// TwinCAT 3 PLC project RedLine3
// ProgramVersion: 3.1.4023.0
// libraries:
//   Tc2_Standard, * (Beckhoff Automation GmbH)
//   Tc2_System, * (Beckhoff Automation GmbH)
//   Tc3_Module, * (Beckhoff Automation GmbH)
// project tree:
//   GVLs/ GVL.TcGVL
//   / PlcTask.TcTTO
//   POUs/ MAIN.TcPOU

CONFIGURATION RedLine3
    RESOURCE PLC ON TwinCAT3
        TASK PlcTask(INTERVAL := T#10ms, PRIORITY := 20);
        PROGRAM MAIN WITH PlcTask : MAIN;
    END_RESOURCE
END_CONFIGURATION

// ---- GVLs/GVL.TcGVL
{attribute 'qualified_only'}
VAR_GLOBAL

//Block States IO
mInSwitch : ARRAY[0..44] OF DINT;
mOutSwitch : ARRAY[0..44] OF DINT;
mInOccupancies : ARRAY[0..44] OF DINT;
mOutOccupancies : ARRAY[0..44] OF DINT;
mInSpeeds : ARRAY[0..44] OF DINT;
mOutSpeeds : ARRAY[0..44] OF DINT;
mInAuthorities : ARRAY[0..44] OF DINT;
mOutAuthorities : ARRAY[0..44] OF DINT;
mInCrossings : ARRAY[0..44] OF DINT;
mOutCrossings : ARRAY[0..44] OF DINT;
mInLeftLights : ARRAY[0..44] OF DINT;
mOutLeftLights : ARRAY[0..44] OF DINT;
mInRightLights : ARRAY[0..44] OF DINT;
mOutRightLights : ARRAY[0..44] OF DINT;
mInMaintenance : ARRAY[0..44] OF DINT;
mOutMaintenance : ARRAY[0..44] OF DINT;
mSpeedLimits : ARRAY[0..44] OF DINT := [40,40,40,40,40,40,40,40,40,40,40,40,40,40,40,40,55,70,70,70,55,55,55,70,70,70,70,70,70,70,70,70,70,70,70,70,70,70,55,55,55,55,55,70];
mInRoute : ARRAY[0..76] OF DINT;
mOutRoute : ARRAY[0..76] OF DINT;


END_VAR

// ---- POUs/MAIN.TcPOU
PROGRAM MAIN
VAR

inc1 : DINT := 0;

	
END_VAR

//0 to 37 map to blocks 1-38
//39 to 44 map to 72-76,yard
//Lights Logic
FOR inc1 := 0 TO 44 DO
	//Sets Red Lights
	IF GVL.mInOccupancies[inc1] = 0
	THEN
		GVL.mOutLeftLights[inc1] := 0;
		GVL.mOutRightLights[inc1] := 0;
	//Sets green lights
	ELSE
		GVL.mOutLeftLights[inc1] := 2;
		GVL.mOutRightLights[inc1] := 2;
	END_IF
END_FOR

FOR inc1 := 1 TO 43 DO
	//Sets Yellow Lights
	IF GVL.mInOccupancies[inc1-1] = 0 AND GVL.mInOccupancies[inc1] <> 0
	THEN
		GVL.mOutRightLights[inc1] := 1;
	END_IF
	IF GVL.mInOccupancies[inc1+1] = 0 AND GVL.mInOccupancies[inc1] <> 0
	THEN
	GVL.mOutLeftLights[inc1] := 1;
	END_IF
END_FOR

//0 to 37 map to blocks 1-38
//39 to 44 map to blocks 72-76,yard
//Passes occupancy, authority, maintenance, and speeds from input to output.
FOR inc1 := 0 TO 44 DO

	GVL.mOutOccupancies[inc1] := GVL.mInOccupancies[inc1];
	GVL.mOutAuthorities[inc1] := GVL.mInAuthorities[inc1];
	GVL.mOutMaintenance[inc1] := GVL.mInMaintenance[inc1];
	IF GVL.mInSpeeds[inc1] < GVL.mSpeedLimits[inc1]
	THEN
		GVL.mOutSpeeds[inc1] := GVL.mInSpeeds[inc1];
	ELSE
		GVL.mOutSpeeds[inc1] := GVL.mSpeedLimits[inc1];
	END_IF
	
END_FOR

FOR inc1 := 0 TO 44 DO

	GVL.mOutRoute[inc1] := GVL.mInRoute[inc1];
	
END_FOR

inc1 := 0;

//This starts the main track logic section

//0 to 37 map to blocks 1-38
//39 to 44 map to 72-76,yard
//Switch Logic
IF GVL.mInMaintenance[8] = 1 
THEN
	IF GVL.mInSwitch[8] = 1
	THEN
		IF GVL.mOutSwitch[8] = 76
		THEN
			GVL.mOutSwitch[8] := 9;
		ELSE
			GVL.mOutSwitch[8] := 76;
		END_IF
		GVL.mInSwitch[8] := 0;
	END_IF
ELSE
    IF GVL.mInOccupancies[44] = 0 
	THEN
    	GVL.mOutSwitch[8] := 76;
    ELSE
		GVL.mOutSwitch[8] := 9;
	END_IF
END_IF

//0 to 37 map to blocks 1-38
//39 to 44 map to 72-76,yard
IF GVL.mInMaintenance[15] = 1 
THEN
    IF GVL.mInSwitch[15] = 1
	THEN
		IF GVL.mOutSwitch[15] = 0
		THEN
			GVL.mOutSwitch[15] := 14;
		ELSE
			GVL.mOutSwitch[15] := 0;
		END_IF
		GVL.mInSwitch[15] := 0;
	END_IF
ELSE
    IF GVL.mInOccupancies[14] = 0 
	THEN
    FOR inc1 := 16 TO 26 DO 
        IF GVL.mInOccupancies[inc1] = 0 
		THEN
            GVL.mOutSwitch[15] := 14;
            Exit;
        ELSE 
            GVL.mOutSwitch[15] := 0;
        END_IF
    END_FOR
	ELSE
		GVL.mOutSwitch[15] := 0;
	END_IF
END_IF

//0 to 37 map to blocks 1-38
//39 to 44 map to 72-76,yard
IF GVL.mInMaintenance[26] = 1 
THEN
    IF GVL.mInSwitch[26] = 1
	THEN
		IF GVL.mOutSwitch[26] = 35
		THEN
			GVL.mOutSwitch[26] := 27;
		ELSE
			GVL.mOutSwitch[26] := 35;
		END_IF
		GVL.mInSwitch[26] := 0;
	END_IF
ELSE
    IF GVL.mInOccupancies[43] = 0 
	THEN
    FOR inc1 := 16 TO 26 DO 
        IF GVL.mInOccupancies[inc1] = 0 
		THEN
            GVL.mOutSwitch[26] := 35;
            Exit;
        ELSE 
            GVL.mOutSwitch[26] := 27;
        END_IF
    END_FOR
	ELSE
		GVL.mOutSwitch[26] := 27;
	END_IF
END_IF

//0 to 37 map to blocks 1-38
//39 to 44 map to 72-76,yard
IF GVL.mInMaintenance[32] = 1 
THEN
    IF GVL.mInSwitch[32] = 1
	THEN
		IF GVL.mOutSwitch[32] = 31
		THEN
			GVL.mOutSwitch[32] := 71;
		ELSE
			GVL.mOutSwitch[32] := 31;
		END_IF
		GVL.mInSwitch[32] := 0;
	END_IF
ELSE
    IF GVL.mInOccupancies[31] = 0 
	THEN
    FOR inc1 := 32 TO 37 DO 
        IF GVL.mInOccupancies[inc1] = 0 
		THEN
            GVL.mOutSwitch[32] := 31;
            Exit;
        ELSE 
            GVL.mOutSwitch[32] := 71;
        END_IF
    END_FOR
	ELSE
		GVL.mOutSwitch[32] := 71;
	END_IF
END_IF

END_PROGRAM
